// TwinCAT 3 PLC project Observer_Pattern
// ProgramVersion: 3.1.4024.0
// libraries:
//   Tc2_Standard, * (Beckhoff Automation GmbH)
//   Tc2_System, * (Beckhoff Automation GmbH)
//   Tc3_Module, * (Beckhoff Automation GmbH)
// project tree:
//   Observers/ Control_Observer.TcPOU, ITF_Observer.TcIO, Motion_Observer.TcPOU
//   / PlcTask.TcTTO
//   POUs/ MAIN.TcPOU
//   Safety/ ITF_TwinSAFEGroup.TcIO, TwinSAFEGroup.TcPOU
// (motion and I/O tree: see PLC project simple_factory_pattern)
// real-time tasks:
//   TASK PlcTask: cycle T#10ms, priority 20, ADS port 350
//   TASK PlcTask1: cycle T#10ms, priority 21, ADS port 351
//   TASK PlcTask2: cycle T#10ms, priority 22, ADS port 352
//   TASK PlcTask3: cycle T#10ms, priority 23, ADS port 353
//   TASK PlcTask4: cycle T#10ms, priority 24, ADS port 354
//   TASK PlcTask5: cycle T#10ms, priority 25, ADS port 355
//   TASK PlcTask6: cycle T#10ms, priority 26, ADS port 356
//   TASK PlcTask7: cycle T#10ms, priority 27, ADS port 357
//   TASK PlcTask8: cycle T#10ms, priority 28, ADS port 358
//   TASK PlcTask9: cycle T#10ms, priority 29, ADS port 359
//   TASK PlcTask10: cycle T#10ms, priority 30, ADS port 360
//   TASK PlcTask11: cycle T#10ms, priority 31, ADS port 361

CONFIGURATION Observer_Pattern
    RESOURCE PLC ON TwinCAT3
        TASK PlcTask(INTERVAL := T#10ms, PRIORITY := 24);
        PROGRAM MAIN WITH PlcTask : MAIN;
    END_RESOURCE
END_CONFIGURATION

// ---- Observers/ITF_Observer.TcIO
INTERFACE ITF_Observer

METHOD Update : BOOL
VAR_INPUT
	TwinSAFEGroup : ITF_TwinSAFEGroup;
END_VAR
END_METHOD

END_INTERFACE

// ---- Safety/ITF_TwinSAFEGroup.TcIO
INTERFACE ITF_TwinSAFEGroup

METHOD GetTwinSAFEState : int
VAR_INPUT
END_VAR
END_METHOD

END_INTERFACE

// ---- POUs/MAIN.TcPOU
PROGRAM MAIN
VAR
	TSGroup : TwinSAFEGroup;
	Control : Control_Observer;
	Motion : Motion_Observer;
	RegisterObservers: BOOL;
END_VAR

IF NOT RegisterObservers THEN
	RegisterObservers := TRUE;
	TSGroup.Subscribe(Control);
	TSGroup.Subscribe(Motion);
END_IF

TSGroup.Cycle();

END_PROGRAM

// ---- Safety/TwinSAFEGroup.TcPOU
FUNCTION_BLOCK TwinSAFEGroup IMPLEMENTS ITF_TwinSAFEGroup
VAR
	MySubscribers : ARRAY[0..9] OF ITF_Observer;
	i: INT;
	SubscriberAlreadyAdded : BOOL;
	NumberOfSubscribers: INT;
	ActTwinSAFEState : INT := 8;
	OldTwinSAFEState : INT;
	Update: BOOL;
END_VAR

METHOD Cycle : BOOL
VAR_INPUT
END_VAR
IF ActTwinSAFEState <> OldTwinSAFEState THEN
	OldTwinSAFEState := ActTwinSAFEState;
	This^.Notify();
END_IF
END_METHOD

METHOD GetTwinSAFEState : INT
VAR_INPUT
END_VAR
GetTwinSAFEState := ActTwinSAFEState;
END_METHOD

METHOD PRIVATE Notify : BOOL
VAR_INPUT
END_VAR
FOR i := 0 TO 9 DO
	IF MySubscribers[i] <> 0 THEN
		MySubscribers[i].Update(THIS^);
	END_IF
END_FOR
END_METHOD

METHOD Subscribe : BOOL
VAR_INPUT
	Subscriber : ITF_Observer;
END_VAR
SubscriberAlreadyAdded := FALSE;
FOR i := 0 TO 9 DO
	IF MySubscribers[i] = Subscriber THEN
		SubscriberAlreadyAdded := TRUE;
	END_IF
END_FOR

IF NOT SubscriberAlreadyAdded THEN
	MySubscribers[NumberOfSubscribers] := Subscriber;
	NumberOfSubscribers := NumberOfSubscribers + 1;
END_IF
END_METHOD

METHOD Unsubscribe : BOOL
VAR_INPUT
	Subscriber : ITF_Observer;
END_VAR
FOR i := 0 TO 9 DO
	IF MySubscribers[i] = Subscriber THEN
		MySubscribers[i] := 0;
		NumberOfSubscribers := NumberOfSubscribers - 1;
	END_IF
END_FOR
END_METHOD

END_FUNCTION_BLOCK

// ---- Observers/Control_Observer.TcPOU
FUNCTION_BLOCK Control_Observer IMPLEMENTS ITF_Observer
VAR
	SystemSafetyState : INT;
END_VAR

METHOD Update : BOOL
VAR_INPUT
	TwinSAFEGroup : ITF_TwinSAFEGroup;
END_VAR
SystemSafetyState := TwinSAFEGroup.GetTwinSAFEState();
END_METHOD

END_FUNCTION_BLOCK

// ---- Observers/Motion_Observer.TcPOU
FUNCTION_BLOCK Motion_Observer IMPLEMENTS ITF_Observer
VAR
	SystemSafetyState : INT;
END_VAR

METHOD Update : BOOL
VAR_INPUT
	TwinSAFEGroup : ITF_TwinSAFEGroup;
END_VAR
SystemSafetyState := TwinSAFEGroup.GetTwinSAFEState();
END_METHOD

END_FUNCTION_BLOCK
